(* Logix 5000 project; controller APM_Relieve Emulate 5570 rev 30.12; software revision 30.00 *)

TASK MainTask (continuous, watchdog 500 ms) : MainProgram

MODULES
   Local : Emulate 5570 (ICP 2, rev 30.12)
      I_O : vendor 1 type 0 code 15 (ICP 3, rev 1.1, Output RPI 50 ms)
END_MODULES

VAR_GLOBAL   (* controller tags *)
   Activa_Maquina_relieve : BOOL := 1;
   ActivarZonaRelieve : BOOL;
   Cuenta_Salida_Acom2 : BOOL;
   EncaminarHorno : BOOL;
   EncaminarRelieve : BOOL;
   Entro_Acom1 : BOOL;
   Entro_Acom2 : BOOL;
   Entro_ParaRelieve : BOOL;
   Entro_ParaRelieve2 : BOOL;
   EstanAdentroAcom2 : BOOL := 1;
   Etapa_Acomodar1 : BOOL;
   EtapaAcomodar2 : BOOL := 1;
   GD_Acomodador1Left1 : BOOL;
   GD_Acomodador1Left2 : BOOL;
   GD_Acomodador2Left1 : BOOL;
   GD_Acomodador2Left2 : BOOL;
   GD_Banda_LLena : BOOL := 1;
   GD_BandaEntradaRelieve1 : BOOL := 1;
   GD_BandaEntradaRelieve2 : BOOL := 1;
   GD_BandaRelieve1 : BOOL := 1;
   GD_BandaRelieve2 : BOOL := 1;
   GD_BandaSalidaRelieve1 : BOOL := 1;
   GD_BandaSalidaRelievePOS : BOOL := 1;
   GD_BandaSalidaRelieveRIGH : BOOL := 1;
   GD_BanEntradaHorno : BOOL := 1;
   GD_BanSalEsmaltado : BOOL := 1;
   GD_Divisor1 : BOOL := 1;
   GD_Divisor2 : BOOL := 1;
   GD_DivisorA : BOOL;
   GD_EntradaRelieveAcomodador1 : BOOL := 1;
   GD_EntradaRelieveAcomodador2 : BOOL := 1;
   GD_IntegradorPos : BOOL := 1;
   GD_IntegradorRIGH : BOOL;
   GD_SalidaAcom2Relieve1 : BOOL := 1;
   GD_SalidaAcom2Relieve2 : BOOL := 1;
   GD_Sens1EntradaAcom2 : BOOL;
   GD_Sens1SalidaAcom1 : BOOL;
   GD_Sens2SalidaAcom1 : BOOL;
   GD_SensDivHorno : BOOL;
   GD_SensDivRelieve : BOOL;
   GD_SensEntradaAcomodador : BOOL;
   GD_SensIntegHorno : BOOL;
   GD_SensIntegRelieve : BOOL;
   GD_SensSalidaAcom2 : BOOL;
   GD_SensSalidaHorno : BOOL;
   GD_VisionSensor1 : DINT;
   IntegrarHorno : BOOL;
   IntegrarRelieve : BOOL;
   IntegrarRelievePrio : BOOL;
   Llego_Acom2 : BOOL;
   LosasAcomodador : COUNTER := (PRE := 3);
   PararLineaRelieve : BOOL;
   Paso_Acom1 : BOOL;
   Paso_Acom2 : COUNTER := (PRE := 4, ACC := 3);
   Paso_ParaHorno : BOOL;
   Paso_ParaRelieve : BOOL;
   Paso_ParaRelieve2 : BOOL;
   PasoSalidaHorno : BOOL;
   PrenderHorno : BOOL := 1;
   RutinaRelieve : BOOL := 1;
   Salida_Relieve : BOOL := 1;
   SensorDivHorno_Down : BOOL;
   SensorDivRelieve_Down : BOOL;
   SensorDivRelieve_Up : BOOL;
   SensorentradaAcom2_UP : BOOL;
   SensorentradaAcomq_Down : BOOL;
   SensorEntroAcom2_Down : BOOL;
   SensorSalidaAcom1_Down : BOOL;
   SensSalidaAcom2_Down : BOOL;
   SensSalidaHorno_Down : BOOL;
   Vision1 : DINT;
END_VAR

PROGRAM MainProgram   (* main routine MainRoutine *)

ROUTINE Entradas   (* ladder *)
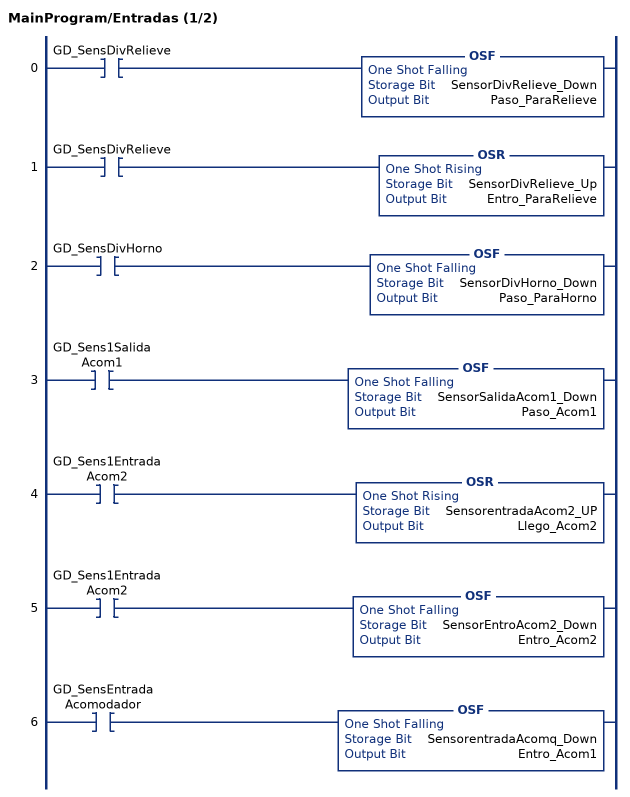
   0: XIC(GD_SensDivRelieve)OSF(SensorDivRelieve_Down,Paso_ParaRelieve);
   1: XIC(GD_SensDivRelieve)OSR(SensorDivRelieve_Up,Entro_ParaRelieve);
   2: XIC(GD_SensDivHorno)OSF(SensorDivHorno_Down,Paso_ParaHorno);
   3: XIC(GD_Sens1SalidaAcom1)OSF(SensorSalidaAcom1_Down,Paso_Acom1);
   4: XIC(GD_Sens1EntradaAcom2)OSR(SensorentradaAcom2_UP,Llego_Acom2);
   5: XIC(GD_Sens1EntradaAcom2)OSF(SensorEntroAcom2_Down,Entro_Acom2);
   6: XIC(GD_SensEntradaAcomodador)OSF(SensorentradaAcomq_Down,Entro_Acom1);
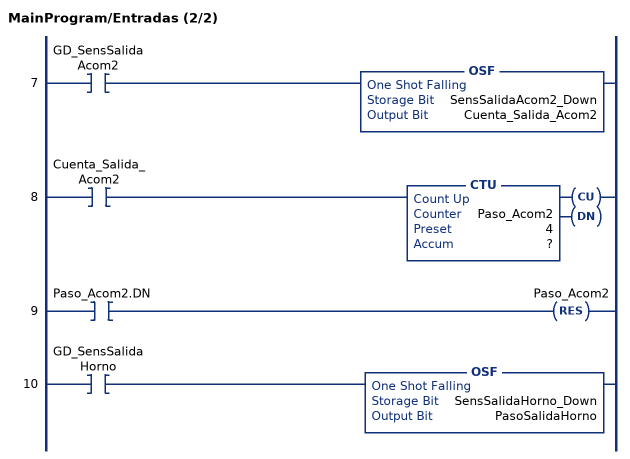
   7: XIC(GD_SensSalidaAcom2)OSF(SensSalidaAcom2_Down,Cuenta_Salida_Acom2);
   8: XIC(Cuenta_Salida_Acom2)CTU(Paso_Acom2,?,?);
   9: XIC(Paso_Acom2.DN)RES(Paso_Acom2);
   10: XIC(GD_SensSalidaHorno)OSF(SensSalidaHorno_Down,PasoSalidaHorno);
END_ROUTINE

ROUTINE IniciarEntrada   (* ladder *)
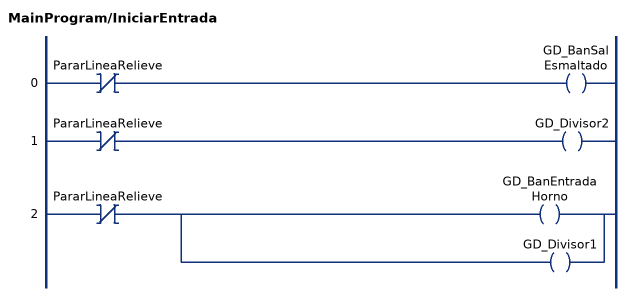
   0: XIO(PararLineaRelieve)OTE(GD_BanSalEsmaltado);
   1: XIO(PararLineaRelieve)OTE(GD_Divisor2);
   2: XIO(PararLineaRelieve)[OTE(GD_BanEntradaHorno) ,OTE(GD_Divisor1) ];
END_ROUTINE

ROUTINE Integrar   (* ladder *)
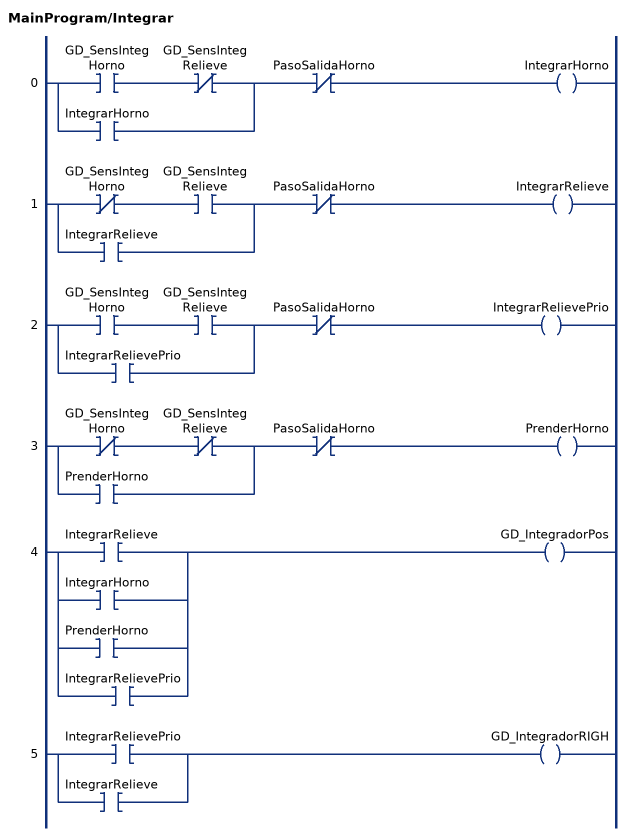
   0: [XIC(GD_SensIntegHorno) XIO(GD_SensIntegRelieve) ,XIC(IntegrarHorno) ]XIO(PasoSalidaHorno)OTE(IntegrarHorno);
   1: [XIO(GD_SensIntegHorno) XIC(GD_SensIntegRelieve) ,XIC(IntegrarRelieve) ]XIO(PasoSalidaHorno)OTE(IntegrarRelieve);
   2: [XIC(GD_SensIntegHorno) XIC(GD_SensIntegRelieve) ,XIC(IntegrarRelievePrio) ]XIO(PasoSalidaHorno)OTE(IntegrarRelievePrio);
   3: [XIO(GD_SensIntegHorno) XIO(GD_SensIntegRelieve) ,XIC(PrenderHorno) ]XIO(PasoSalidaHorno)OTE(PrenderHorno);
   4: [XIC(IntegrarRelieve) ,[XIC(IntegrarHorno) ,[XIC(PrenderHorno) ,XIC(IntegrarRelievePrio) ] ] ]OTE(GD_IntegradorPos);
   5: [XIC(IntegrarRelievePrio) ,XIC(IntegrarRelieve) ]OTE(GD_IntegradorRIGH);
END_ROUTINE

ROUTINE MainRoutine   (* ladder *)
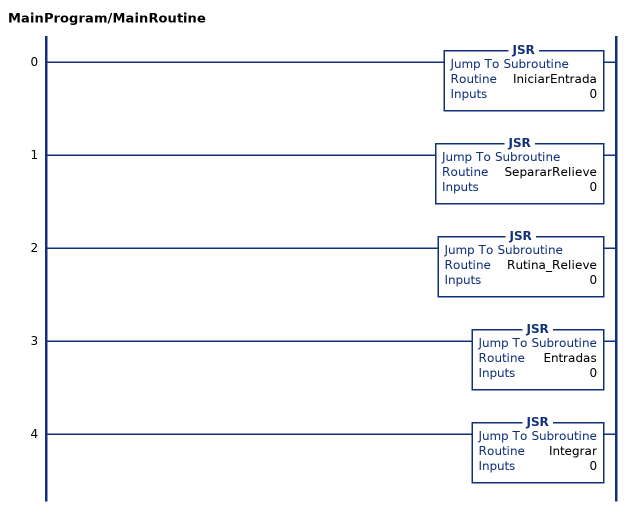
   0: JSR(IniciarEntrada,0);
   1: JSR(SepararRelieve,0);
   2: JSR(Rutina_Relieve,0);
   3: JSR(Entradas,0);
   4: JSR(Integrar,0);
END_ROUTINE

ROUTINE Rutina_Relieve   (* ladder *)
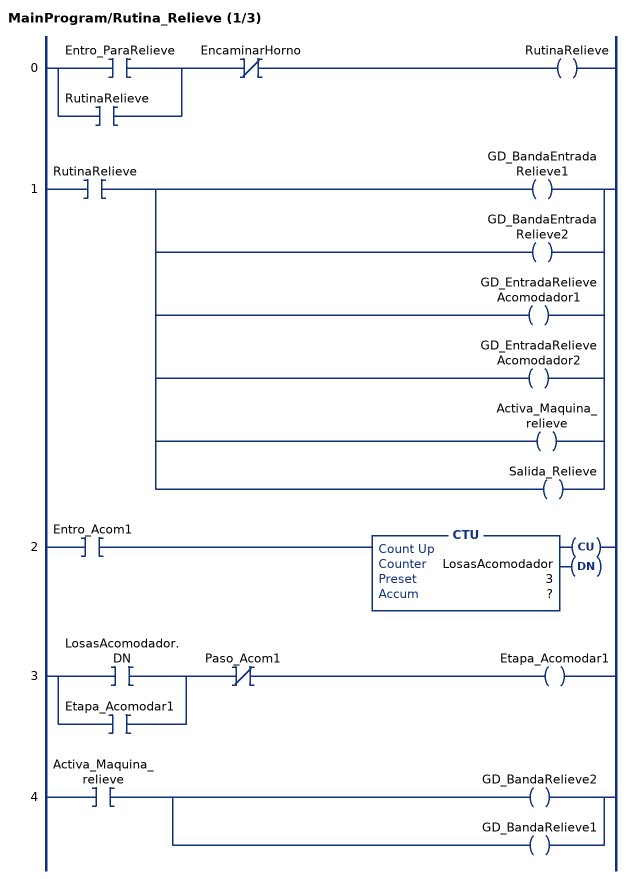
   0: [XIC(Entro_ParaRelieve) ,XIC(RutinaRelieve) ]XIO(EncaminarHorno)OTE(RutinaRelieve);
   1: XIC(RutinaRelieve)[OTE(GD_BandaEntradaRelieve1) ,[OTE(GD_BandaEntradaRelieve2) ,[OTE(GD_EntradaRelieveAcomodador1) ,[OTE(GD_EntradaRelieveAcomodador2) ,[OTE(Activa_Maquina_relieve) ,OTE(Salida_Relieve) ] ] ] ] ];
   2: XIC(Entro_Acom1)CTU(LosasAcomodador,?,?);
   3: [XIC(LosasAcomodador.DN) ,XIC(Etapa_Acomodar1) ]XIO(Paso_Acom1)OTE(Etapa_Acomodar1);
   4: XIC(Activa_Maquina_relieve)[OTE(GD_BandaRelieve2) ,OTE(GD_BandaRelieve1) ];
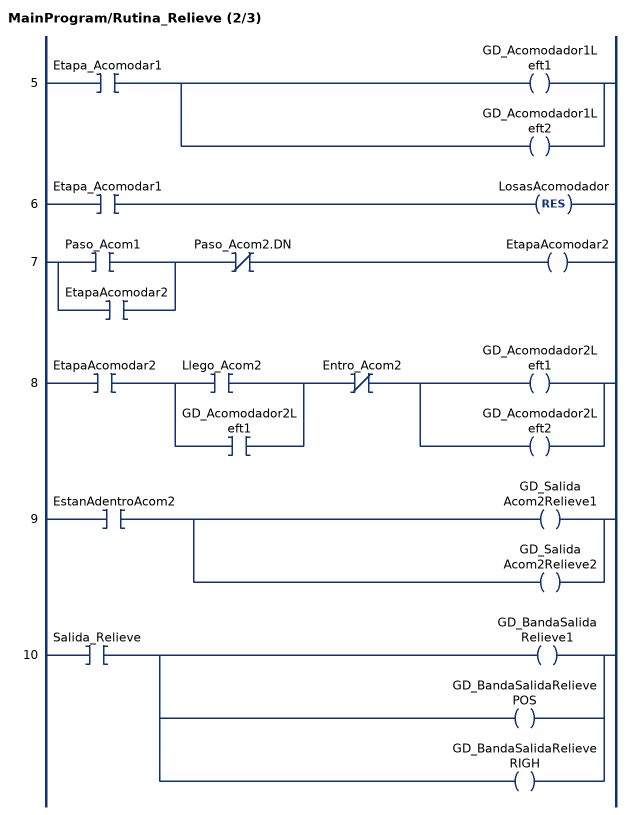
   5: XIC(Etapa_Acomodar1)[OTE(GD_Acomodador1Left1) ,OTE(GD_Acomodador1Left2) ];
   6: XIC(Etapa_Acomodar1)RES(LosasAcomodador);
   7: [XIC(Paso_Acom1) ,XIC(EtapaAcomodar2) ]XIO(Paso_Acom2.DN)OTE(EtapaAcomodar2);
   8: XIC(EtapaAcomodar2)[XIC(Llego_Acom2) ,XIC(GD_Acomodador2Left1) ]XIO(Entro_Acom2)[OTE(GD_Acomodador2Left1) ,OTE(GD_Acomodador2Left2) ];
   9: XIC(EstanAdentroAcom2)[OTE(GD_SalidaAcom2Relieve1) ,OTE(GD_SalidaAcom2Relieve2) ];
   10: XIC(Salida_Relieve)[OTE(GD_BandaSalidaRelieve1) ,[OTE(GD_BandaSalidaRelievePOS) ,OTE(GD_BandaSalidaRelieveRIGH) ] ];
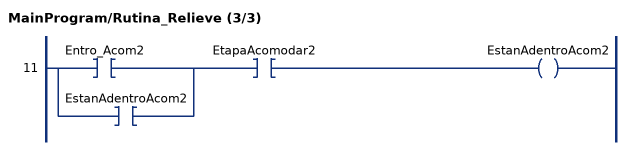
   11: [XIC(Entro_Acom2) ,XIC(EstanAdentroAcom2) ]XIC(EtapaAcomodar2)OTE(EstanAdentroAcom2);
END_ROUTINE

ROUTINE SepararRelieve   (* ladder *)
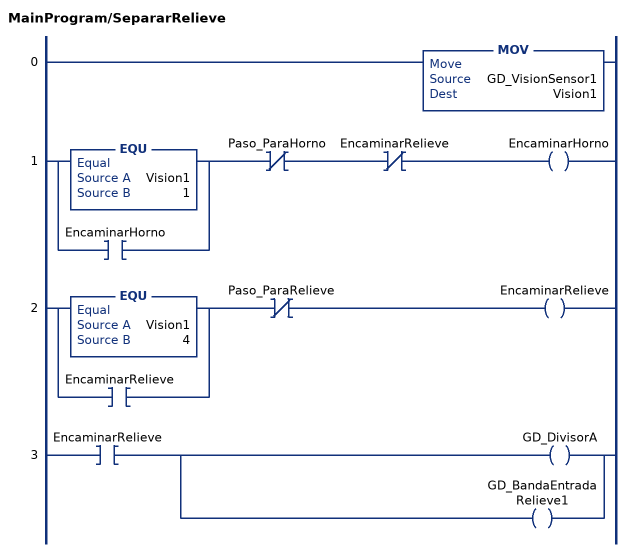
   0: MOV(GD_VisionSensor1,Vision1);
   1: [EQU(Vision1,1) ,XIC(EncaminarHorno) ]XIO(Paso_ParaHorno)XIO(EncaminarRelieve)OTE(EncaminarHorno);
   2: [EQU(Vision1,4) ,XIC(EncaminarRelieve) ]XIO(Paso_ParaRelieve)OTE(EncaminarRelieve);
   3: XIC(EncaminarRelieve)[OTE(GD_DivisorA) ,OTE(GD_BandaEntradaRelieve1) ];
END_ROUTINE
END_PROGRAM
